FUNCTION_BLOCK trip_timer (* Basic Function Block Type *)
  (* Standard: 61499-2 *)
  (* Version 0.0, 11/29/2016, gulzha, nxtControl GmbH, Template *)
  PACKAGE Main;
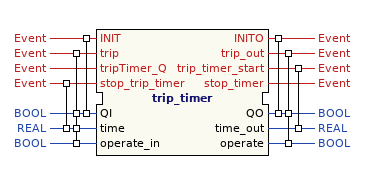
  EVENT_INPUT
    INIT WITH QI; (* Initialization Request *)
    trip WITH QI, time, operate_in; (* Normal Execution Request *)
    tripTimer_Q;
    stop_trip_timer WITH time;
  END_EVENT
  EVENT_OUTPUT
    INITO WITH QO; (* Initialization Confirm *)
    trip_out WITH QO, operate; (* Execution Confirmation *)
    trip_timer_start WITH time_out;
    stop_timer;
  END_EVENT
  VAR_INPUT
    QI : BOOL; (* Input event qualifier *)
    time : REAL;
    operate_in : BOOL;
  END_VAR
  VAR_OUTPUT
    QO : BOOL; (* Output event qualifier *)
    time_out : REAL;
    operate : BOOL;
  END_VAR
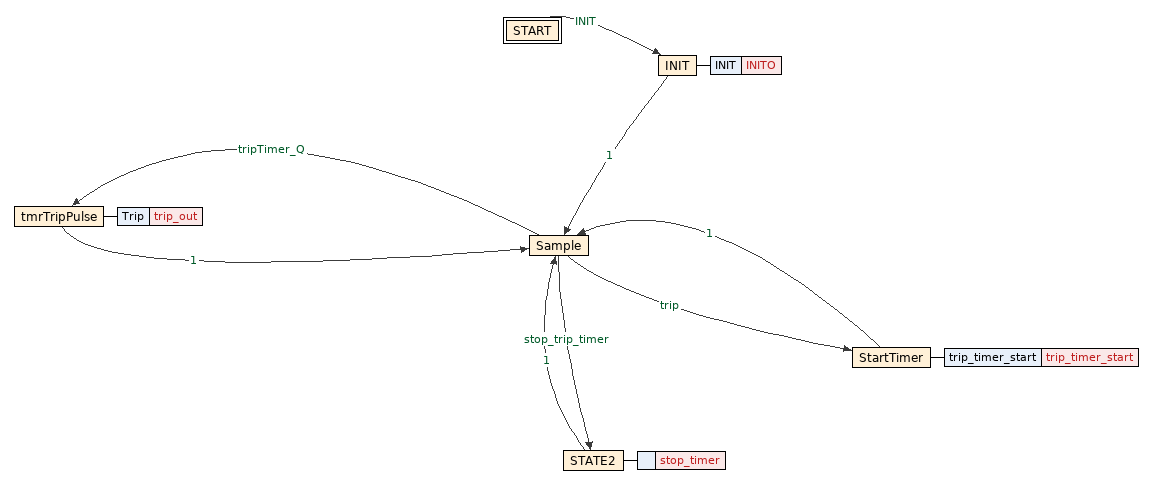
  EC_STATES
    START; (* Initial State *)
    INIT : INIT -> INITO; (* Initialization *)
    Sample;
    tmrTripPulse : Trip -> trip_out;
    StartTimer : trip_timer_start -> trip_timer_start;
    STATE2 : -> stop_timer;
  END_STATES
  EC_TRANSITIONS
    INIT TO Sample := 1;
    Sample TO tmrTripPulse := tripTimer_Q;
    StartTimer TO Sample := 1;
    tmrTripPulse TO Sample := 1;
    START TO INIT := INIT;
    Sample TO StartTimer := trip;
    Sample TO STATE2 := stop_trip_timer;
    STATE2 TO Sample := 1;
  END_TRANSITIONS
  ALGORITHM INIT IN ST: (* Initialization algorithm *)
;
operate := FALSE;
operate_in := FALSE;
  END_ALGORITHM
  ALGORITHM REQ IN ST: (* Normally executed algorithm *)
;
  END_ALGORITHM
  ALGORITHM trip_timer_start IN ST:
;
time_out := time;
  END_ALGORITHM
  ALGORITHM reset_pulse_internal IN ST:
;
operate := FALSE;
time_out:=0;
  END_ALGORITHM
  ALGORITHM trip_pulse_timer IN ST:
;
  END_ALGORITHM
  ALGORITHM Trip IN ST:
;
//operate := TRUE;
operate := operate_in;
  END_ALGORITHM
  ALGORITHM setVar IN ST:
;
  END_ALGORITHM
END_FUNCTION_BLOCK
